TYPE ST_2DPoint :
STRUCT
	X : REAL;	//X Koordinate in µm
	Y : REAL;	//X Koordinate in µm	
END_STRUCT
END_TYPE

(* stored: Version 1.1.0.1, ProductVersion 3.1.0.25
   DUT ST_2DPoint: Id {b97bb7b3-c261-4f31-88ea-0251ea187d61} *)
